// TIA Portal V17 export
// export: Created 2022-07-05T08:45:16.725064Z, ExportSetting WithDefaults, DisplayName Totally Integrated Automation Portal, DisplayVersion V17, DisplayName TIA Portal Openness, DisplayVersion V17, DisplayName TIA Portal Version Control Interface, DisplayVersion V17, DisplayName STEP 7 Professional, DisplayVersion V17, DisplayName STEP 7 Safety, DisplayVersion V17, DisplayName WinCC Advanced, DisplayVersion V17
DATA_BLOCK "InstOpcUaClient"   // DB3
VERSION : 0.1
// stored: AutoNumber true, DBAccessibleFromOPCUA true, DBAccessibleFromWebserver true, InstanceOfName OpcUaClient, InstanceOfType FB
"OpcUaClient"
   // VAR_INPUT
   //    enable : Bool;
   //    read : Bool;
   //    write : Bool;
   //    callMethod : Bool;
   //    methodHdlIndex : SInt;
   //    connectionInfo : OPC_UA_SessionConnectInfo;
   //    serverEndpointUrl : String;
   // END_VAR
   // VAR_OUTPUT
   //    connected { ExternalWritable := 'False'} : Bool;
   //    done { ExternalWritable := 'False'} : Bool;
   //    busy { ExternalWritable := 'False'} : Bool;
   //    error { ExternalWritable := 'False'} : Bool;
   //    status { ExternalWritable := 'False'} : Word;
   //    diagnostics { ExternalWritable := 'False'} : "typeFbDiagnostics";
   //    connectionHdl { ExternalWritable := 'False'} : DWord;
   // END_VAR
   // VAR_IN_OUT
   //    namespaceUris : Variant;
   //    namespaceIndexes : Variant;
   //    readNodeIds : Variant;
   //    readNodeHdls : Variant;
   //    readData : Variant;
   //    writeNodeIds : Variant;
   //    writeNodeHdls : Variant;
   //    writeData : Variant;
   //    objNodeIds : Variant;
   //    methodNodeIds : Variant;
   //    methodHdls : Variant;
   //    inputArguments : Variant;
   //    outputArguments : Variant;
   // END_VAR
   // VAR
   //    instOpcUaConnect { ExternalAccessible := 'False'; ExternalVisible := 'False'; ExternalWritable := 'False'; S7_SetPoint := 'True'} : OPC_UA_Connect;
   //    instOpcUaConnectionGetStatus { ExternalAccessible := 'False'; ExternalVisible := 'False'; ExternalWritable := 'False'; S7_SetPoint := 'True'} : OPC_UA_ConnectionGetStatus;
   //    instOpcUaNamespaceGIL { ExternalAccessible := 'False'; ExternalVisible := 'False'; ExternalWritable := 'False'; S7_SetPoint := 'True'} : OPC_UA_NamespaceGetIndexList;
   //    InstOpcUaGHLRead { ExternalAccessible := 'False'; ExternalVisible := 'False'; ExternalWritable := 'False'; S7_SetPoint := 'True'} : OPC_UA_NodeGetHandleList;
   //    instOpcUaGHLWrite { ExternalAccessible := 'False'; ExternalVisible := 'False'; ExternalWritable := 'False'; S7_SetPoint := 'True'} : OPC_UA_NodeGetHandleList;
   //    instOpcUaGHLMethods { ExternalAccessible := 'False'; ExternalVisible := 'False'; ExternalWritable := 'False'; S7_SetPoint := 'True'} : OPC_UA_MethodGetHandleList;
   //    InstOpcUaRHLRead { ExternalAccessible := 'False'; ExternalVisible := 'False'; ExternalWritable := 'False'; S7_SetPoint := 'True'} : OPC_UA_NodeReleaseHandleList;
   //    instOpcUaRHLWrite { ExternalAccessible := 'False'; ExternalVisible := 'False'; ExternalWritable := 'False'; S7_SetPoint := 'True'} : OPC_UA_NodeReleaseHandleList;
   //    instOpcUaRHLMethods { ExternalAccessible := 'False'; ExternalVisible := 'False'; ExternalWritable := 'False'; S7_SetPoint := 'True'} : OPC_UA_MethodReleaseHandleList;
   //    instOpcUaReadList { ExternalAccessible := 'False'; ExternalVisible := 'False'; ExternalWritable := 'False'; S7_SetPoint := 'True'} : OPC_UA_ReadList;
   //    instOpcUaWriteList { ExternalAccessible := 'False'; ExternalVisible := 'False'; ExternalWritable := 'False'; S7_SetPoint := 'True'} : OPC_UA_WriteList;
   //    instOpcUaMethodCall { ExternalAccessible := 'False'; ExternalVisible := 'False'; ExternalWritable := 'False'; S7_SetPoint := 'True'} : OPC_UA_MethodCall;
   //    instOpcUaDisconnect { ExternalAccessible := 'False'; ExternalVisible := 'False'; ExternalWritable := 'False'; S7_SetPoint := 'True'} : OPC_UA_Disconnect;
   //    statOldTriggers { ExternalAccessible := 'False'; ExternalVisible := 'False'; ExternalWritable := 'False'} : Struct
   //       connect { ExternalAccessible := 'False'; ExternalVisible := 'False'; ExternalWritable := 'False'} : Bool;
   //       reconnect { ExternalAccessible := 'False'; ExternalVisible := 'False'; ExternalWritable := 'False'} : Bool;
   //       disconnect { ExternalAccessible := 'False'; ExternalVisible := 'False'; ExternalWritable := 'False'; S7_SetPoint := 'True'} : Bool;
   //       read { ExternalAccessible := 'False'; ExternalVisible := 'False'; ExternalWritable := 'False'; S7_SetPoint := 'True'} : Bool;
   //       write { ExternalAccessible := 'False'; ExternalVisible := 'False'; ExternalWritable := 'False'; S7_SetPoint := 'True'} : Bool;
   //       callMethod { ExternalAccessible := 'False'; ExternalVisible := 'False'; ExternalWritable := 'False'} : Bool;
   //       clearSession { ExternalAccessible := 'False'; ExternalVisible := 'False'; ExternalWritable := 'False'} : Bool;
   //    END_STRUCT;
   //    statState { ExternalWritable := 'False'} : Int;
   //    statDone { ExternalAccessible := 'False'; ExternalVisible := 'False'; ExternalWritable := 'False'} : Bool;
   //    statConnected { ExternalAccessible := 'False'; ExternalVisible := 'False'; ExternalWritable := 'False'} : Bool;
   //    statBusy { ExternalVisible := 'False'; ExternalWritable := 'False'} : Bool;
   //    statDiagnostics { ExternalAccessible := 'False'; ExternalVisible := 'False'; ExternalWritable := 'False'; S7_SetPoint := 'True'} : "typeFbDiagnostics";
   //    statDiagnosticsEmpty { ExternalWritable := 'False'; S7_SetPoint := 'True'} : "typeFbDiagnostics";
   //    statOpcUaRequests { ExternalAccessible := 'False'; ExternalVisible := 'False'; ExternalWritable := 'False'} : Struct
   //       connect { ExternalAccessible := 'False'; ExternalVisible := 'False'; ExternalWritable := 'False'} : Bool;
   //       conGS { ExternalAccessible := 'False'; ExternalVisible := 'False'; ExternalWritable := 'False'} : Bool;
   //       NGIL { ExternalAccessible := 'False'; ExternalVisible := 'False'; ExternalWritable := 'False'} : Bool;
   //       readGHL { ExternalAccessible := 'False'; ExternalVisible := 'False'; ExternalWritable := 'False'} : Bool;
   //       methodsGHL { ExternalAccessible := 'False'; ExternalVisible := 'False'; ExternalWritable := 'False'} : Bool;
   //       writeGHL { ExternalAccessible := 'False'; ExternalVisible := 'False'; ExternalWritable := 'False'} : Bool;
   //       read { ExternalAccessible := 'False'; ExternalVisible := 'False'; ExternalWritable := 'False'} : Bool;
   //       write { ExternalAccessible := 'False'; ExternalVisible := 'False'; ExternalWritable := 'False'} : Bool;
   //       methodCall { ExternalAccessible := 'False'; ExternalVisible := 'False'; ExternalWritable := 'False'} : Bool;
   //       readRHL { ExternalAccessible := 'False'; ExternalVisible := 'False'; ExternalWritable := 'False'} : Bool;
   //       writeRHL { ExternalAccessible := 'False'; ExternalVisible := 'False'; ExternalWritable := 'False'} : Bool;
   //       methodsRHL { ExternalAccessible := 'False'; ExternalVisible := 'False'; ExternalWritable := 'False'} : Bool;
   //       disconnect { ExternalAccessible := 'False'; ExternalVisible := 'False'; ExternalWritable := 'False'} : Bool;
   //    END_STRUCT;
   //    statRegisteredLists { ExternalWritable := 'False'} : Struct
   //       NamespaceIndexes { ExternalWritable := 'False'} : Bool;
   //       Read { ExternalWritable := 'False'} : Bool;
   //       Write { ExternalWritable := 'False'} : Bool;
   //       Methods { ExternalWritable := 'False'} : Bool;
   //    END_STRUCT;
   //    statDiagCounter { ExternalWritable := 'False'} : Struct
   //       Connect { ExternalVisible := 'False'; ExternalWritable := 'False'} : UInt;
   //       NamespaceReg { ExternalWritable := 'False'} : UInt;
   //       RegisterRead { ExternalWritable := 'False'} : UInt;
   //       RegisterWrite { ExternalWritable := 'False'} : UInt;
   //       RegisterMethods { ExternalWritable := 'False'} : UInt;
   //       Read { ExternalWritable := 'False'} : UInt;
   //       Write { ExternalWritable := 'False'} : UInt;
   //       MethodCall { ExternalWritable := 'False'} : UInt;
   //    END_STRUCT;
   //    statMethodResult { ExternalWritable := 'False'} : DWord;
   //    statMethodHdl { ExternalAccessible := 'False'; ExternalVisible := 'False'; ExternalWritable := 'False'} : DWord;
   //    statMethodHdlId { ExternalAccessible := 'False'; ExternalVisible := 'False'; ExternalWritable := 'False'} : DInt;
   //    statConnectionHdl { ExternalAccessible := 'False'; ExternalVisible := 'False'; ExternalWritable := 'False'} : DWord;
   //    statRHLTrigger { ExternalAccessible := 'False'; ExternalVisible := 'False'; ExternalWritable := 'False'} : Bool;
   //    statCheckConnectionStatus { ExternalAccessible := 'False'; ExternalVisible := 'False'; ExternalWritable := 'False'} : Bool;
   //    statCycDiagTrigger { ExternalAccessible := 'False'; ExternalVisible := 'False'; ExternalWritable := 'False'} : Bool;
   //    instCycDiag { ExternalAccessible := 'False'; ExternalVisible := 'False'; ExternalWritable := 'False'; S7_SetPoint := 'True'} : IEC_TIMER;
   //    statOpcUaReadTimeStamps { ExternalWritable := 'False'} : Array[0..299] of LDT;
   //    statSerializeMethodHdls { ExternalAccessible := 'False'; ExternalVisible := 'False'; ExternalWritable := 'False'} : Array[0..1199] of Byte;
   //    statOpcUaStatusLists { ExternalWritable := 'False'} : Struct
   //       methodRHL { ExternalWritable := 'False'} : Array[0..299] of DWord;
   //       methodGHL { ExternalWritable := 'False'} : Array[0..299] of DWord;
   //       writeRHL { ExternalWritable := 'False'} : Array[0..299] of DWord;
   //       writeList { ExternalWritable := 'False'} : Array[0..299] of DWord;
   //       writeGHL { ExternalWritable := 'False'} : Array[0..299] of DWord;
   //       readRHL { ExternalWritable := 'False'} : Array[0..299] of DWord;
   //       readList { ExternalWritable := 'False'} : Array[0..299] of DWord;
   //       readGHL { ExternalWritable := 'False'} : Array[0..299] of DWord;
   //       namespaceGIL { ExternalWritable := 'False'} : Array[0..299] of DWord;
   //    END_STRUCT;
   // END_VAR
BEGIN
END_DATA_BLOCK
